FUNCTION_BLOCK FB_SendAutoPilotFlag_Right
VAR_INPUT
	AutoPilotFlag : INT;
END_VAR
VAR_OUTPUT
END_VAR
VAR
	TxMessage : EXTCANQUEUE;
END_VAR
VAR_IN_OUT
	CAN_OUTPUTS_Right : CANTXQUEUESTRUCT_E_32;
	CAN_INPUTS_Right : CANRXQUEUESTRUCT_E_32;
END_VAR

 
TxMessage.cobId := 130;
TxMessage.length := 1;
TxMessage.data[0] :=  INT_TO_BYTE(AutoPilotFlag AND 16#FF);
CAN_OUTPUTS_Right.TxMessages[11] := TxMessage;
//CAN_OUTPUTS.NoOfTxMessages := 1;

END_FUNCTION_BLOCK

(* stored: Version 1.1.0.1
   POU FB_SendAutoPilotFlag_Right: Id {c069e083-877e-4f96-9eb0-ad9ca255ef75}, SpecialFunc None *)
